FUNCTION_BLOCK Sensor_Merge2 (* Basic FB with empty ECC *)
  (* Standard: 61499-2 *)
  (* Version 1.0, 2023-03-02, AK125171 *)
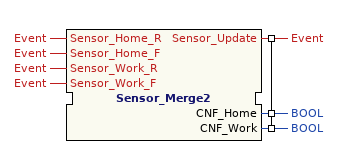
  EVENT_INPUT
    Sensor_Home_R;
    Sensor_Home_F;
    Sensor_Work_R;
    Sensor_Work_F;
  END_EVENT
  EVENT_OUTPUT
    Sensor_Update WITH CNF_Home, CNF_Work;
  END_EVENT
  VAR_OUTPUT
    CNF_Home : BOOL;
    CNF_Work : BOOL;
  END_VAR
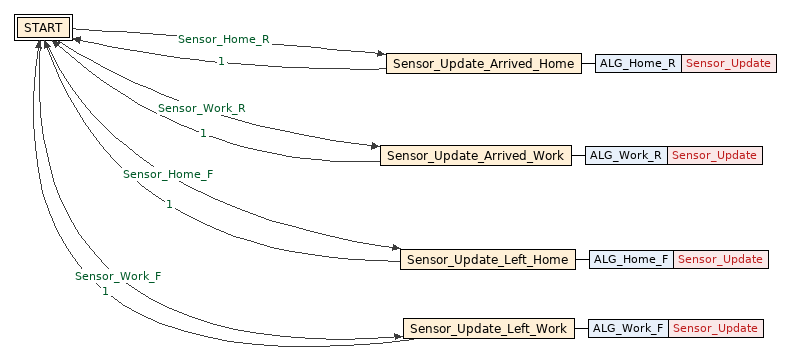
  EC_STATES
    START; (* Initial State *)
    Sensor_Update_Arrived_Home : ALG_Home_R -> Sensor_Update;
    Sensor_Update_Arrived_Work : ALG_Work_R -> Sensor_Update;
    Sensor_Update_Left_Home : ALG_Home_F -> Sensor_Update;
    Sensor_Update_Left_Work : ALG_Work_F -> Sensor_Update;
  END_STATES
  EC_TRANSITIONS
    START TO Sensor_Update_Arrived_Home := Sensor_Home_R;
    START TO Sensor_Update_Arrived_Work := Sensor_Work_R;
    Sensor_Update_Arrived_Home TO START := 1;
    Sensor_Update_Arrived_Work TO START := 1;
    START TO Sensor_Update_Left_Home := Sensor_Home_F;
    Sensor_Update_Left_Home TO START := 1;
    START TO Sensor_Update_Left_Work := Sensor_Work_F;
    Sensor_Update_Left_Work TO START := 1;
  END_TRANSITIONS
  ALGORITHM ALG_Work_R IN ST:
CNF_Work:=TRUE;
CNF_Home:=FALSE;
  END_ALGORITHM
  ALGORITHM ALG_Home_R IN ST:
CNF_Home:=TRUE;
CNF_Work:=FALSE;
  END_ALGORITHM
  ALGORITHM ALG_Home_F IN ST:
CNF_Home:=FALSE;
CNF_Work:=FALSE;
  END_ALGORITHM
  ALGORITHM ALG_Work_F IN ST:
CNF_Work:=FALSE;
CNF_Home:=FALSE;
  END_ALGORITHM
END_FUNCTION_BLOCK
